// TIA Portal project "Phiva_v4" (V17)

(* hardware
DEVICE "S71500/ET200MP station_1"  S7-1500 station
   slot 0: "Rail_0"  Rack  6ES7 590-1***0-0AA0
   slot 1: "station_1"  CPU 1512C-1 PN  6ES7 512-1CK01-0AB0  V2.5
      slot 3: "CPU display_1"  6ES7591-1AA00-0AA0
      slot 32768: "PROFINET interface_1"  X1
         slot 32769: "Port_1"  X1 P1
         slot 32770: "Port_2"  X1 P2
DEVICE "S71500/ET200MP station_2"  S7-1500 station
   slot 0: "Rail_0"  Rack  6ES7 590-1***0-0AA0
   slot 1: "station_2"  CPU 1512C-1 PN  6ES7 512-1CK01-0AB0  V2.5
      slot 3: "CPU display_1"  6ES7591-1AA00-0AA0
      slot 32768: "PROFINET interface_1"  X1
         slot 32769: "Port_1"  X1 P1
         slot 32770: "Port_2"  X1 P2
DEVICE "HMI_1"  TP700 Comfort
   slot 0: "HMI_1"  TP700 Comfort  6AV2 124-0GC01-0AX0  15.0.0.0
   slot 1: "HMI_RT_1"  TP700 Comfort  6AV2 124-0GC01-0AX0  15.0.0.0
   slot 5: "HMI_1.IE_CP_1"  PROFINET Interface  15.0.0.0
      slot 1: "PROFINET Interface_1"  PROFINET Interface
         slot 1: "Port_1"  Port
         slot 2: "Port_2"  Port
   slot 7: "HMI_1.MPI/DP_CP_1"  MPI/DP Interface  15.0.0.0
*)

// ===== PLC "station_1"  CPU 1512C-1 PN =====

VAR_GLOBAL   // PLC tag table "Default tag table"
   "START" AT %I10.0 : Bool;
   "STOP" AT %I10.1 : Bool;
   "AUTO" AT %I10.2 : Bool;
   "RESET" AT %I10.3 : Bool;
   "START LED" AT %Q4.0 : Bool;
   "RESET LED" AT %Q4.1 : Bool;
   "Q1 LED" AT %Q4.2 : Bool;
   "Q2 LED" AT %Q4.3 : Bool;
   "4 EXTEND PUSH CYLINDER" AT %Q5.4 : Bool;
   "reset_timer_delay_bit" AT %M0.1 : Bool;
   "6 CONVEYOR_1_FORWARD" AT %Q5.0 : Bool;
   "8 INDUCTIVE SENSOR (NO)metal" AT %I11.2 : Bool;
   "7 PART AT DETECTION POSITION(NO)" AT %I11.1 : Bool;
   "5 PUSH CYLINDER EXTENDED" AT %I11.7 : Bool;
   "3 PART IN MAGAZINE (NC)" AT %I11.6 : Bool;
   "power_on_mem" AT %M0.0 : Bool;
   "9 PART AT END CONVEYOR (NO)" AT %I11.0 : Bool;
   "conveyor 2 set active mem" AT %M110.0 : Bool;
   "Tag_1" AT %M200.0 : Bool;
   "System_Byte" AT %MB1 : Byte;
   "FirstScan" AT %M1.0 : Bool;
   "DiagStatusUpdate" AT %M1.1 : Bool;
   "AlwaysTRUE" AT %M1.2 : Bool;
   "AlwaysFALSE" AT %M1.3 : Bool;
   "Clock_Byte" AT %MB500 : Byte;
   "Clock_10Hz" AT %M500.0 : Bool;
   "Clock_5Hz" AT %M500.1 : Bool;
   "Clock_2.5Hz" AT %M500.2 : Bool;
   "Clock_2Hz" AT %M500.3 : Bool;
   "Clock_1.25Hz" AT %M500.4 : Bool;
   "Clock_1Hz" AT %M500.5 : Bool;
   "Clock_0.625Hz" AT %M500.6 : Bool;
   "Clock_0.5Hz" AT %M500.7 : Bool;
   "metal sensor info" AT %M60.0 : Bool;
   "end of conveyor 1" AT %M60.1 : Bool;
   "metal sensor info int" AT %IW60 : Int;
   "any wkpiece info" AT %M80.0 : Bool;
   "station 2 end status" AT %M80.1 : Bool;
   "Tag_2" AT %M70.2 : Bool;
END_VAR

DATA_BLOCK "Data_block_1"   // DB1
{ S7_Optimized_Access := 'FALSE' }
VERSION : 0.1
   VAR
      start_bit : Bool;
      stop_bit : Bool;
      reset_bit : Bool;
      manual_set_bit : Bool;
      power_on_mem : Bool;
      "system_active?" : Bool;
      process_no : Word;
      time_preset : Time := T#2_500MS;
      monitering_time : Time;
      "metal sensor info" : Bool;
      "conveyor 2 status" : Bool;
      "metal sensor info int" : Int;
   END_VAR
BEGIN
END_DATA_BLOCK

DATA_BLOCK "GET"   // DB15
{ S7_Optimized_Access := 'TRUE' }
VERSION : 0.1
   VAR
      GET : Bool;
   END_VAR
BEGIN
END_DATA_BLOCK

// folder: System blocks/Program resources

DATA_BLOCK "reset_button_timer1"   // DB2
{ S7_Optimized_Access := 'TRUE' }
AUTHOR : Simatic
FAMILY : IEC
NAME : IEC_TMR
VERSION : 1.0
// stored: InstanceOfName IEC_TIMER
"IEC_TIMER"
BEGIN
END_DATA_BLOCK

DATA_BLOCK "IEC_Timer_0_DB_2"   // DB3
{ S7_Optimized_Access := 'TRUE' }
AUTHOR : Simatic
FAMILY : IEC
NAME : IEC_TMR
VERSION : 1.0
// stored: InstanceOfName IEC_TIMER
"IEC_TIMER"
BEGIN
END_DATA_BLOCK

DATA_BLOCK "reset_button_timer2"   // DB4
{ S7_Optimized_Access := 'TRUE' }
AUTHOR : Simatic
FAMILY : IEC
NAME : IEC_TMR
VERSION : 1.0
// stored: InstanceOfName IEC_TIMER
"IEC_TIMER"
BEGIN
END_DATA_BLOCK

DATA_BLOCK "IEC_Counter_0_DB"   // DB5
{ S7_Optimized_Access := 'TRUE' }
AUTHOR : Simatic
FAMILY : IEC
NAME : CNTR
VERSION : 1.0
// stored: InstanceOfName IEC_COUNTER
"IEC_COUNTER"
BEGIN
END_DATA_BLOCK

DATA_BLOCK "IEC_Timer_0_DB_3"   // DB6
{ S7_Optimized_Access := 'TRUE' }
AUTHOR : Simatic
FAMILY : IEC
NAME : IEC_TMR
VERSION : 1.0
// stored: InstanceOfName IEC_TIMER
"IEC_TIMER"
BEGIN
END_DATA_BLOCK

DATA_BLOCK "IEC_Counter_0_DB_1"   // DB7
{ S7_Optimized_Access := 'TRUE' }
AUTHOR : Simatic
FAMILY : IEC
NAME : CNTR
VERSION : 1.0
// stored: InstanceOfName IEC_COUNTER
"IEC_COUNTER"
BEGIN
END_DATA_BLOCK

DATA_BLOCK "IEC_Counter_0_DB_2"   // DB8
{ S7_Optimized_Access := 'TRUE' }
AUTHOR : Simatic
FAMILY : IEC
NAME : CNTR
VERSION : 1.0
// stored: InstanceOfName IEC_COUNTER
"IEC_COUNTER"
BEGIN
END_DATA_BLOCK

DATA_BLOCK "reset_time_latch_countdown1"   // DB10
{ S7_Optimized_Access := 'TRUE' }
AUTHOR : Simatic
FAMILY : IEC
NAME : IEC_TMR
VERSION : 1.0
// stored: InstanceOfName IEC_TIMER
"IEC_TIMER"
BEGIN
END_DATA_BLOCK

DATA_BLOCK "IEC_Timer_0_DB"   // DB13
{ S7_Optimized_Access := 'TRUE' }
AUTHOR : Simatic
FAMILY : IEC
NAME : IEC_TMR
VERSION : 1.0
// stored: InstanceOfName IEC_TIMER
"IEC_TIMER"
BEGIN
END_DATA_BLOCK

DATA_BLOCK "IEC_Timer_0_DB_1"   // DB14
{ S7_Optimized_Access := 'TRUE' }
AUTHOR : Simatic
FAMILY : IEC
NAME : IEC_TMR
VERSION : 1.0
// stored: InstanceOfName IEC_TIMER
"IEC_TIMER"
BEGIN
END_DATA_BLOCK

// folder: (top level)

FUNCTION "Auto_Mode" : Void   // FC1, LAD
{ S7_Optimized_Access := 'TRUE' }
VERSION : 0.1
   VAR_TEMP   // added for the SCL form of the ladder/FBD networks
      _w1 : Bool;
      _w2 : Bool;
   END_VAR
BEGIN

REGION Network 1: Detection of material at entry
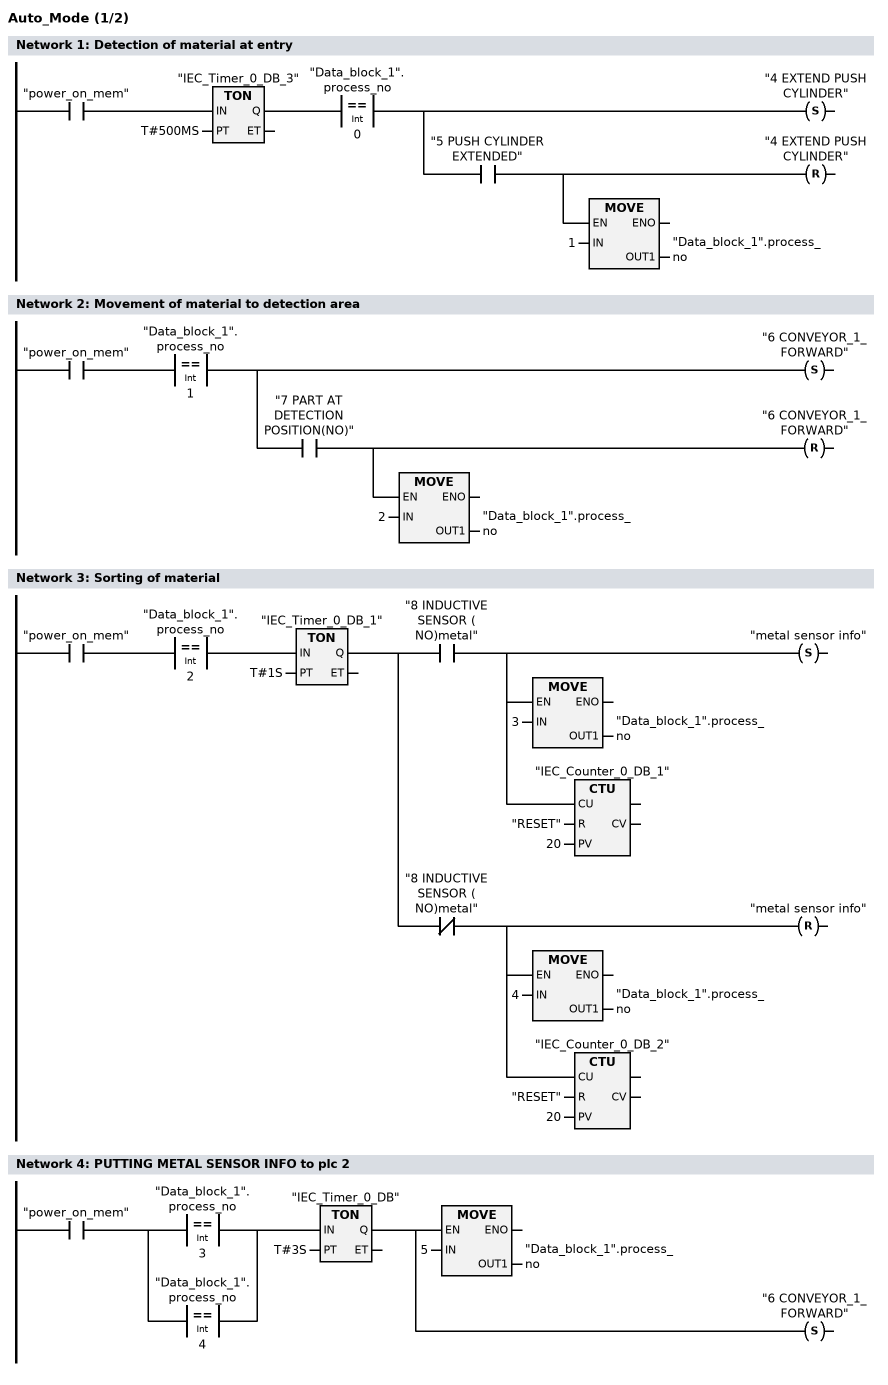
   "IEC_Timer_0_DB_3".TON(IN := "power_on_mem", PT := T#500MS);
   #_w1 := "IEC_Timer_0_DB_3".Q AND ("Data_block_1".process_no = 0);
   IF #_w1 THEN "4 EXTEND PUSH CYLINDER" := TRUE; END_IF;
   IF #_w1 AND "5 PUSH CYLINDER EXTENDED" THEN
       "4 EXTEND PUSH CYLINDER" := FALSE;
       "Data_block_1".process_no := 1;
   END_IF;
END_REGION

REGION Network 2: Movement of material to detection area
   RUNG wire#powerrail
      Contact( "power_on_mem" )
      { S7_Templates := "SrcType := Int" } EQ_Contact(in1 := "Data_block_1".process_no, in2 := 1)
      wire#w1
      S_Coil( "6 CONVEYOR_1_FORWARD" )
   END_RUNG
   RUNG wire#w1
      Contact( "7 PART AT DETECTION POSITION(NO)" )
      wire#w2
      R_Coil( "6 CONVEYOR_1_FORWARD" )
   END_RUNG
   RUNG wire#w2
      Move(in := 2, out1 => "Data_block_1".process_no)
   END_RUNG
   // the same network as SCL:
   #_w1 := "power_on_mem" AND ("Data_block_1".process_no = 1);
   IF #_w1 THEN "6 CONVEYOR_1_FORWARD" := TRUE; END_IF;
   IF #_w1 AND "7 PART AT DETECTION POSITION(NO)" THEN
       "6 CONVEYOR_1_FORWARD" := FALSE;
       "Data_block_1".process_no := 2;
   END_IF;
END_REGION

REGION Network 3: Sorting of material
   "IEC_Timer_0_DB_1".TON(IN := "power_on_mem" AND ("Data_block_1".process_no = 2), PT := T#1S);
   #_w1 := "IEC_Timer_0_DB_1".Q AND "8 INDUCTIVE SENSOR (NO)metal";
   IF #_w1 THEN
       "metal sensor info" := TRUE;
       "Data_block_1".process_no := 3;
   END_IF;
   "IEC_Counter_0_DB_1".CTU(CU := #_w1, R := "RESET", PV := 20);
   #_w2 := "IEC_Timer_0_DB_1".Q AND NOT "8 INDUCTIVE SENSOR (NO)metal";
   IF #_w2 THEN
       "metal sensor info" := FALSE;
       "Data_block_1".process_no := 4;
   END_IF;
   "IEC_Counter_0_DB_2".CTU(CU := #_w2, R := "RESET", PV := 20);
END_REGION

REGION Network 4: PUTTING METAL SENSOR INFO to plc 2
   "IEC_Timer_0_DB".TON(IN := "power_on_mem" AND (("Data_block_1".process_no = 3) OR ("Data_block_1".process_no = 4)),
                        PT := T#3S);
   IF "IEC_Timer_0_DB".Q THEN
       "Data_block_1".process_no := 5;
       "6 CONVEYOR_1_FORWARD" := TRUE;
   END_IF;
END_REGION

REGION Network 5: End of conveyor 1
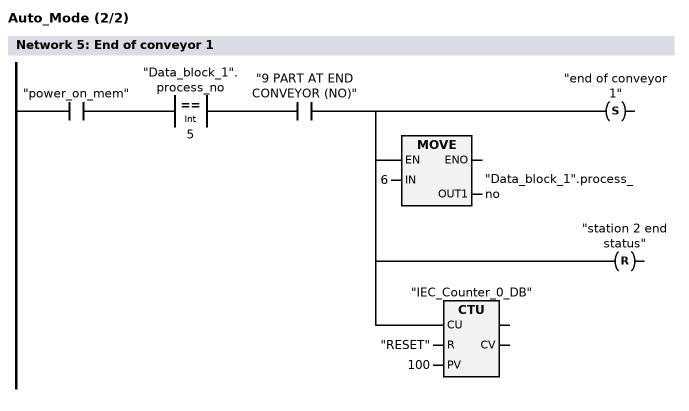
   #_w1 := "power_on_mem" AND ("Data_block_1".process_no = 5) AND "9 PART AT END CONVEYOR (NO)";
   IF #_w1 THEN
       "end of conveyor 1" := TRUE;
       "Data_block_1".process_no := 6;
       "station 2 end status" := FALSE;
   END_IF;
   "IEC_Counter_0_DB".CTU(CU := #_w1, R := "RESET", PV := 100);
END_REGION
END_FUNCTION

FUNCTION "Manual_Mode" : Void   // FC2, LAD
{ S7_Optimized_Access := 'TRUE' }
VERSION : 0.1
BEGIN
END_FUNCTION

ORGANIZATION_BLOCK "Main"   // OB1, LAD, ProgramCycle
TITLE = "Main Program Sweep (Cycle)"
{ S7_Optimized_Access := 'TRUE' }
VERSION : 0.1
   VAR_INPUT
      Initial_Call : Bool;   // Initial call of this OB
      Remanence : Bool;   // =True, if remanent data are available
   END_VAR
   VAR_TEMP   // added for the SCL form of the ladder/FBD networks
      _w1 : Bool;
   END_VAR
BEGIN

REGION Network 1: POWER MEM
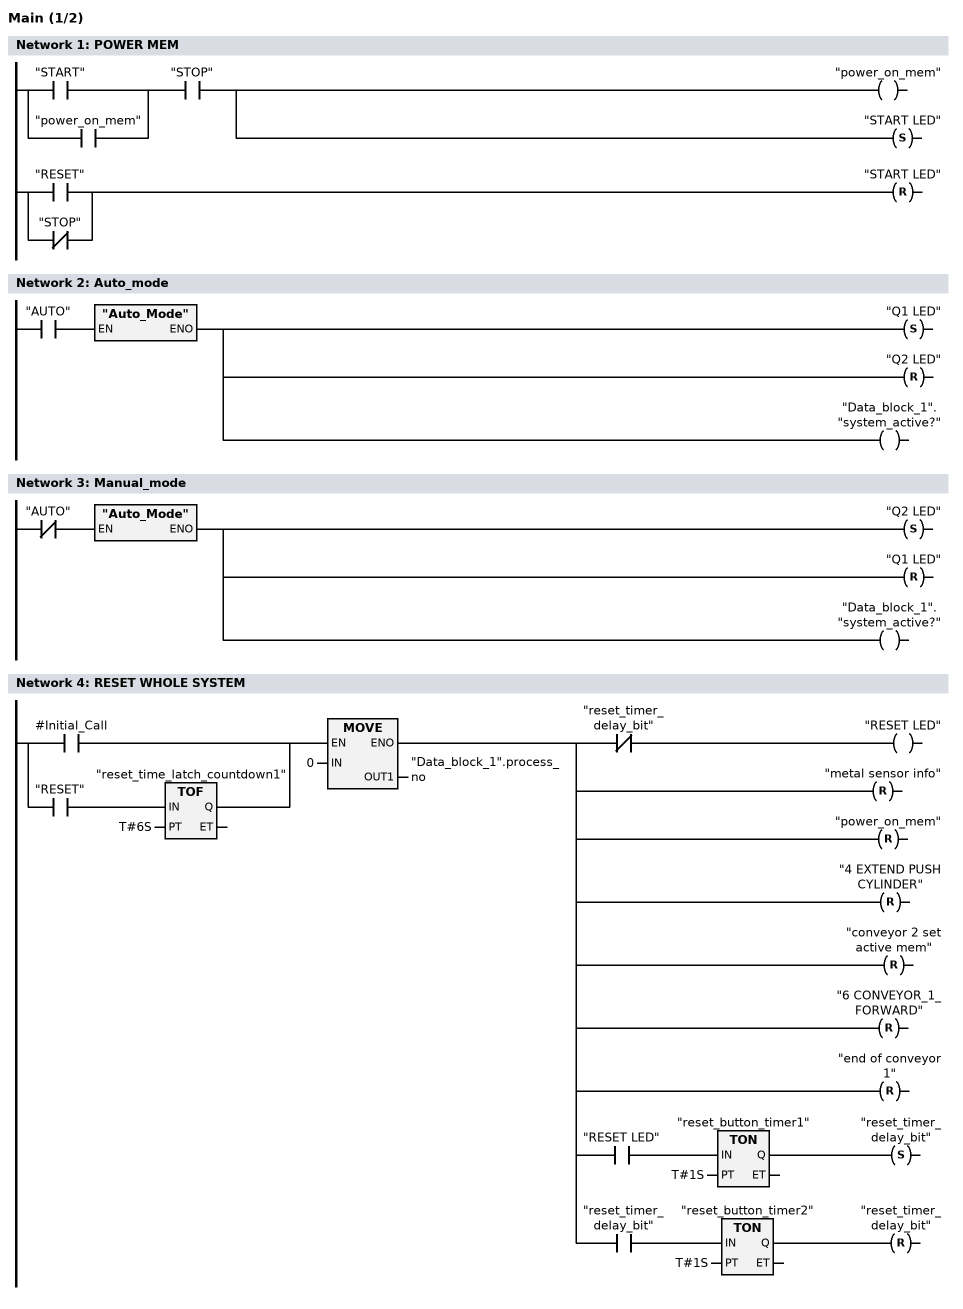
   RUNG wire#powerrail
      Contact( "START" )
      wire#w1
      Contact( "STOP" )
      wire#w2
      Coil( "power_on_mem" )
   END_RUNG
   RUNG wire#powerrail
      Contact( "power_on_mem" )
   END_RUNG wire#w1
   RUNG wire#w2
      S_Coil( "START LED" )
   END_RUNG
   RUNG wire#powerrail
      Contact( "RESET" )
      wire#w3
      R_Coil( "START LED" )
   END_RUNG
   RUNG wire#powerrail
      I_Contact( "STOP" )
   END_RUNG wire#w3
   // the same network as SCL:
   "power_on_mem" := ("START" OR "power_on_mem") AND "STOP";
   IF "power_on_mem" THEN "START LED" := TRUE; END_IF;
   IF "RESET" OR NOT "STOP" THEN "START LED" := FALSE; END_IF;
END_REGION

REGION Network 2: Auto_mode
   RUNG wire#powerrail
      Contact( "AUTO" )
      "Auto_Mode"()
      wire#w1
      S_Coil( "Q1 LED" )
   END_RUNG
   RUNG wire#w1
      R_Coil( "Q2 LED" )
   END_RUNG
   RUNG wire#w1
      Coil( "Data_block_1"."system_active?" )
   END_RUNG
   // the same network as SCL:
   "Auto_Mode"(EN := "AUTO", ENO => #_w1);
   IF #_w1 THEN
       "Q1 LED" := TRUE;
       "Q2 LED" := FALSE;
   END_IF;
   "Data_block_1"."system_active?" := #_w1;
END_REGION

REGION Network 3: Manual_mode
   RUNG wire#powerrail
      I_Contact( "AUTO" )
      "Auto_Mode"()
      wire#w1
      S_Coil( "Q2 LED" )
   END_RUNG
   RUNG wire#w1
      R_Coil( "Q1 LED" )
   END_RUNG
   RUNG wire#w1
      Coil( "Data_block_1"."system_active?" )
   END_RUNG
   // the same network as SCL:
   "Auto_Mode"(EN := NOT "AUTO", ENO => #_w1);
   IF #_w1 THEN
       "Q2 LED" := TRUE;
       "Q1 LED" := FALSE;
   END_IF;
   "Data_block_1"."system_active?" := #_w1;
END_REGION

REGION Network 4: RESET WHOLE SYSTEM
   "reset_time_latch_countdown1".TOF(IN := "RESET", PT := T#6S);
   #_w1 := #Initial_Call OR "reset_time_latch_countdown1".Q;
   IF #_w1 THEN "Data_block_1".process_no := 0; END_IF;
   "RESET LED" := #_w1 AND NOT "reset_timer_delay_bit";
   IF #_w1 THEN
       "metal sensor info" := FALSE;
       "power_on_mem" := FALSE;
       "4 EXTEND PUSH CYLINDER" := FALSE;
       "conveyor 2 set active mem" := FALSE;
       "6 CONVEYOR_1_FORWARD" := FALSE;
       "end of conveyor 1" := FALSE;
   END_IF;
   "reset_button_timer1".TON(IN := #_w1 AND "RESET LED", PT := T#1S);
   IF "reset_button_timer1".Q THEN "reset_timer_delay_bit" := TRUE; END_IF;
   "reset_button_timer2".TON(IN := #_w1 AND "reset_timer_delay_bit", PT := T#1S);
   IF "reset_button_timer2".Q THEN "reset_timer_delay_bit" := FALSE; END_IF;
END_REGION

REGION Network 5: get data from plc 2
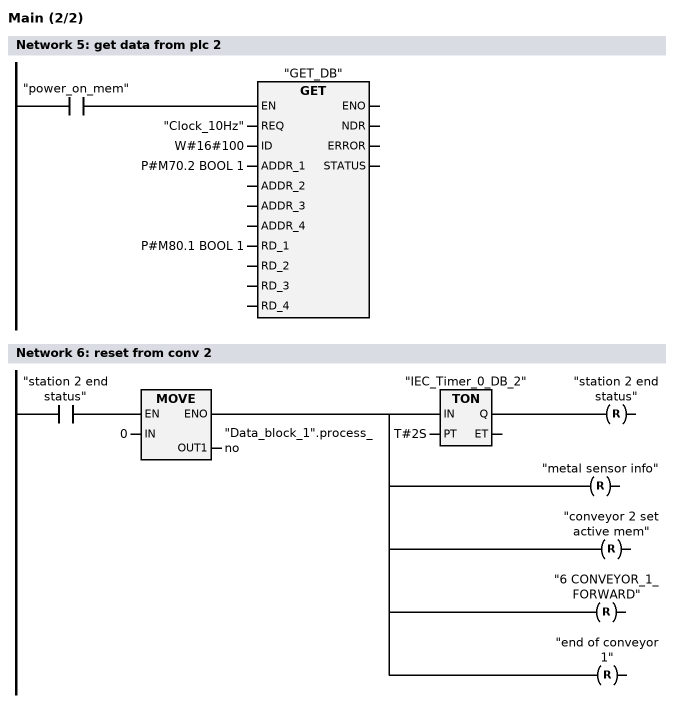
   IF "power_on_mem" THEN
       "GET_DB"(REQ := "Clock_10Hz", ID := W#16#100, ADDR_1 := P#M70.2 BOOL 1, RD_1 := P#M80.1 BOOL 1);   // GET
   END_IF;
END_REGION

REGION Network 6: reset from conv 2
   IF "station 2 end status" THEN "Data_block_1".process_no := 0; END_IF;
   "IEC_Timer_0_DB_2".TON(IN := "station 2 end status", PT := T#2S);
   #_w1 := "station 2 end status";
   IF "IEC_Timer_0_DB_2".Q THEN "station 2 end status" := FALSE; END_IF;
   IF #_w1 THEN
       "metal sensor info" := FALSE;
       "conveyor 2 set active mem" := FALSE;
       "6 CONVEYOR_1_FORWARD" := FALSE;
       "end of conveyor 1" := FALSE;
   END_IF;
END_REGION
END_ORGANIZATION_BLOCK

// ===== PLC "station_2"  CPU 1512C-1 PN =====

VAR_GLOBAL   // PLC tag table "Default tag table"
   "START (NO)" AT %I10.0 : Bool;
   "STOP (NC)" AT %I10.1 : Bool;
   "AUTO" AT %I10.2 : Bool;
   "RESET" AT %I10.3 : Bool;
   "START LED" AT %Q4.0 : Bool;
   "RESET LED" AT %Q4.1 : Bool;
   "Q1 LED" AT %Q4.2 : Bool;
   "Q2 LED" AT %Q4.3 : Bool;
   "8 CONVEYOR 3 FORWARD" AT %Q6.0 : Bool;
   "5 WORKPIECE AT CONVEYOR 2 BARRIER (NC)" AT %I12.0 : Bool;
   "6 CALL ROBOT FOR 2 SEC" AT %Q6.4 : Bool;
   "7 ROBOT DROPPED WORKPIECE AT CONVEYOR 3 (NO)" AT %I12.4 : Bool;
   "9 WORKPIECE EXITING  CONVEYOR 3 (NO)" AT %I12.2 : Bool;
   "3 CONVEYOR 2 FORWARD" AT %Q6.3 : Bool;
   "4 CONVEYOR 2 BARRIER" AT %Q6.2 : Bool;
   "power_on_mem" AT %M0.0 : Bool;
   "6.1 WORKPIECE EXITING STATION 2 (NO)" AT %I12.1 : Bool;
   "non-metal_or_metal_info from plc 1" AT %M70.0 : Bool;
   "Clock_Byte" AT %MB600 : Byte;
   "Clock_10Hz" AT %M600.0 : Bool;
   "Clock_5Hz" AT %M600.1 : Bool;
   "Clock_2.5Hz" AT %M600.2 : Bool;
   "Clock_2Hz" AT %M600.3 : Bool;
   "Clock_1.25Hz" AT %M600.4 : Bool;
   "Clock_1Hz" AT %M600.5 : Bool;
   "Clock_0.625Hz" AT %M600.6 : Bool;
   "Clock_0.5Hz" AT %M600.7 : Bool;
   "reset_timer_delay_bit" AT %M20.0 : Bool;
   "metal sensor info" AT %M20.1 : Bool;
   "conveyor 2 set active mem" AT %M20.2 : Bool;
   "Tag_1" AT %M60.1 : Bool;
   "workpiece ready" AT %M70.1 : Bool;
   "conveyor 2 end process" AT %M70.2 : Bool;
END_VAR

DATA_BLOCK "Receive_data_Block_1"   // DB2
{ S7_Optimized_Access := 'FALSE' }
VERSION : 0.1
   VAR
      "non-metal_or_metal_info" : Bool;
   END_VAR
BEGIN
END_DATA_BLOCK

DATA_BLOCK "Data_block_1"   // DB4
{ S7_Optimized_Access := 'FALSE' }
VERSION : 0.1
   VAR
      process_no : Word;
   END_VAR
BEGIN
END_DATA_BLOCK

// folder: System blocks/Program resources

DATA_BLOCK "IEC_Timer_0_DB"   // DB3
{ S7_Optimized_Access := 'TRUE' }
AUTHOR : Simatic
FAMILY : IEC
NAME : IEC_TMR
VERSION : 1.0
// stored: InstanceOfName IEC_TIMER
"IEC_TIMER"
BEGIN
END_DATA_BLOCK

DATA_BLOCK "IEC_Timer_0_DB_1"   // DB5
{ S7_Optimized_Access := 'TRUE' }
AUTHOR : Simatic
FAMILY : IEC
NAME : IEC_TMR
VERSION : 1.0
// stored: InstanceOfName IEC_TIMER
"IEC_TIMER"
BEGIN
END_DATA_BLOCK

DATA_BLOCK "IEC_Timer_0_DB_2"   // DB6
{ S7_Optimized_Access := 'TRUE' }
AUTHOR : Simatic
FAMILY : IEC
NAME : IEC_TMR
VERSION : 1.0
// stored: InstanceOfName IEC_TIMER
"IEC_TIMER"
BEGIN
END_DATA_BLOCK

DATA_BLOCK "IEC_Counter_0_DB"   // DB7
{ S7_Optimized_Access := 'TRUE' }
AUTHOR : Simatic
FAMILY : IEC
NAME : CNTR
VERSION : 1.0
// stored: InstanceOfName IEC_COUNTER
"IEC_COUNTER"
BEGIN
END_DATA_BLOCK

DATA_BLOCK "IEC_Timer_0_DB_3"   // DB8
{ S7_Optimized_Access := 'TRUE' }
AUTHOR : Simatic
FAMILY : IEC
NAME : IEC_TMR
VERSION : 1.0
// stored: InstanceOfName IEC_TIMER
"IEC_TIMER"
BEGIN
END_DATA_BLOCK

DATA_BLOCK "IEC_Timer_0_DB_4"   // DB9
{ S7_Optimized_Access := 'TRUE' }
AUTHOR : Simatic
FAMILY : IEC
NAME : IEC_TMR
VERSION : 1.0
// stored: InstanceOfName IEC_TIMER
"IEC_TIMER"
BEGIN
END_DATA_BLOCK

DATA_BLOCK "IEC_Counter_0_DB_1"   // DB10
{ S7_Optimized_Access := 'TRUE' }
AUTHOR : Simatic
FAMILY : IEC
NAME : CNTR
VERSION : 1.0
// stored: InstanceOfName IEC_COUNTER
"IEC_COUNTER"
BEGIN
END_DATA_BLOCK

DATA_BLOCK "IEC_Timer_0_DB_5"   // DB11
{ S7_Optimized_Access := 'TRUE' }
AUTHOR : Simatic
FAMILY : IEC
NAME : IEC_TMR
VERSION : 1.0
// stored: InstanceOfName IEC_TIMER
"IEC_TIMER"
BEGIN
END_DATA_BLOCK

DATA_BLOCK "IEC_Timer_0_DB_6"   // DB12
{ S7_Optimized_Access := 'TRUE' }
AUTHOR : Simatic
FAMILY : IEC
NAME : IEC_TMR
VERSION : 1.0
// stored: InstanceOfName IEC_TIMER
"IEC_TIMER"
BEGIN
END_DATA_BLOCK

// folder: (top level)

FUNCTION "Auto_mode_plc_2" : Void   // FC1, LAD
{ S7_Optimized_Access := 'TRUE' }
VERSION : 0.1
   VAR_TEMP   // added for the SCL form of the ladder/FBD networks
      _w1 : Bool;
      _w2 : Bool;
   END_VAR
BEGIN

REGION Network 1: workpiece in conveyor 2
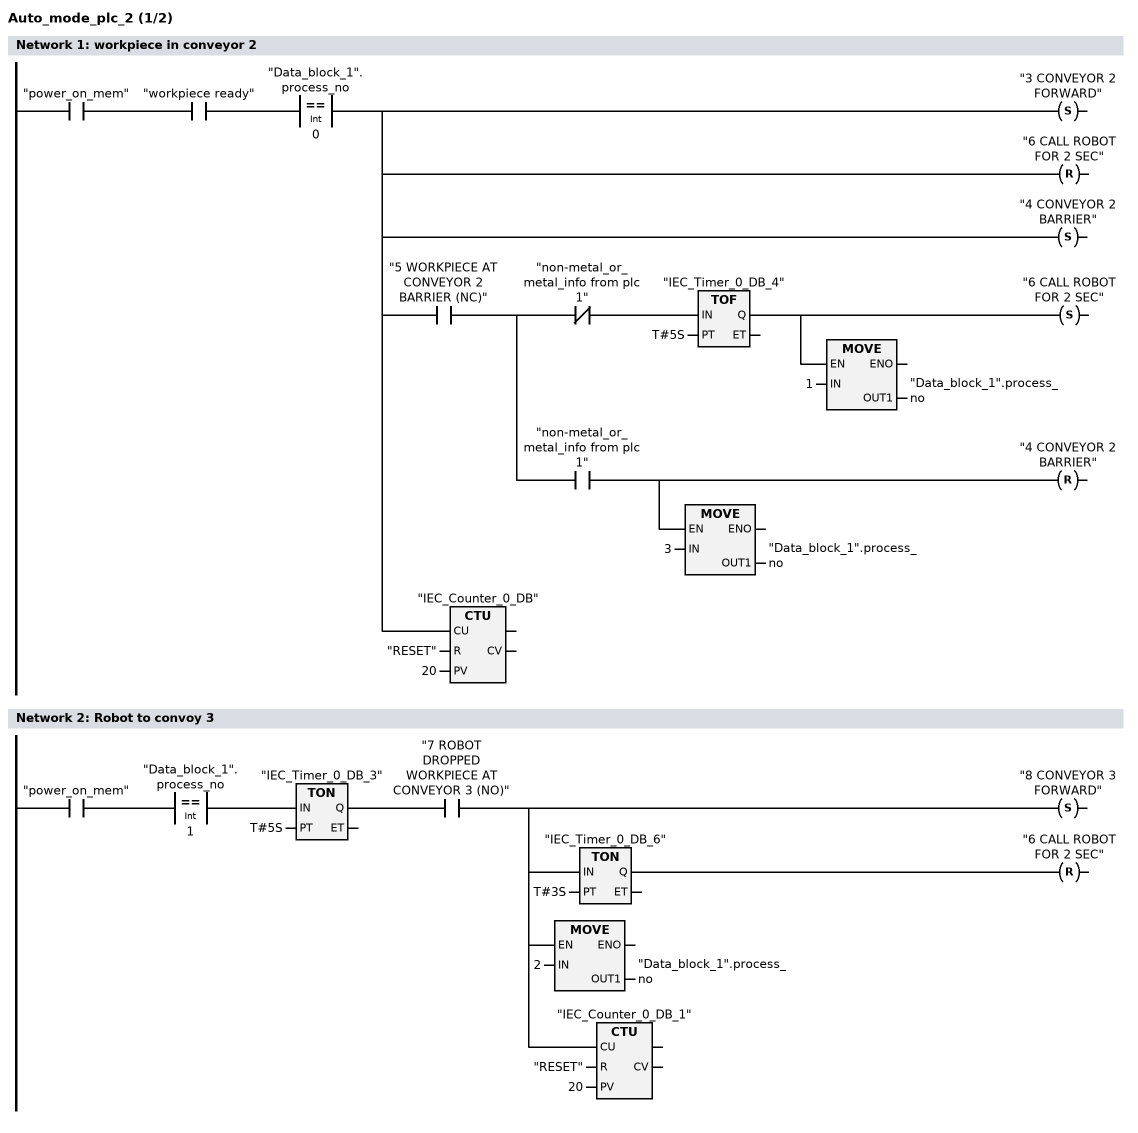
   #_w1 := "power_on_mem" AND "workpiece ready" AND ("Data_block_1".process_no = 0);
   IF #_w1 THEN
       "3 CONVEYOR 2 FORWARD" := TRUE;
       "6 CALL ROBOT FOR 2 SEC" := FALSE;
       "4 CONVEYOR 2 BARRIER" := TRUE;
   END_IF;
   #_w2 := #_w1 AND "5 WORKPIECE AT CONVEYOR 2 BARRIER (NC)";
   "IEC_Timer_0_DB_4".TOF(IN := #_w2 AND NOT "non-metal_or_metal_info from plc 1", PT := T#5S);
   IF "IEC_Timer_0_DB_4".Q THEN
       "6 CALL ROBOT FOR 2 SEC" := TRUE;
       "Data_block_1".process_no := 1;
   END_IF;
   IF #_w2 AND "non-metal_or_metal_info from plc 1" THEN
       "4 CONVEYOR 2 BARRIER" := FALSE;
       "Data_block_1".process_no := 3;
   END_IF;
   "IEC_Counter_0_DB".CTU(CU := #_w1, R := "RESET", PV := 20);
END_REGION

REGION Network 2: Robot to convoy 3
   "IEC_Timer_0_DB_3".TON(IN := "power_on_mem" AND ("Data_block_1".process_no = 1), PT := T#5S);
   #_w1 := "IEC_Timer_0_DB_3".Q AND "7 ROBOT DROPPED WORKPIECE AT CONVEYOR 3 (NO)";
   IF #_w1 THEN "8 CONVEYOR 3 FORWARD" := TRUE; END_IF;
   "IEC_Timer_0_DB_6".TON(IN := #_w1, PT := T#3S);
   IF "IEC_Timer_0_DB_6".Q THEN "6 CALL ROBOT FOR 2 SEC" := FALSE; END_IF;
   IF #_w1 THEN "Data_block_1".process_no := 2; END_IF;
   "IEC_Counter_0_DB_1".CTU(CU := #_w1, R := "RESET", PV := 20);
END_REGION

REGION Network 3: Metal convoyor 3 end + Non-metal exiting station 2
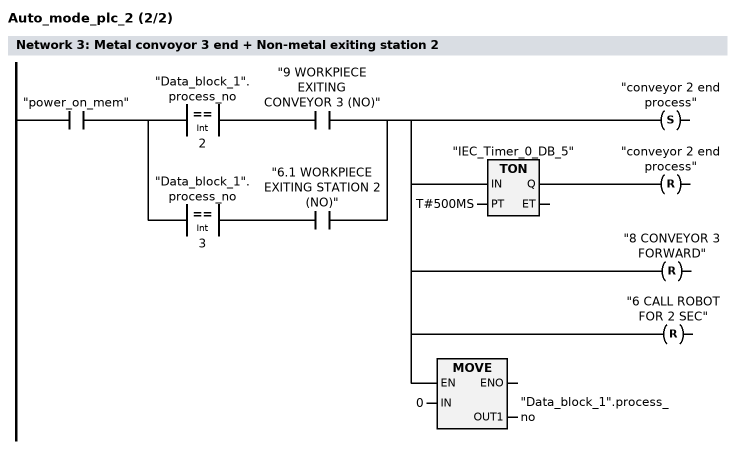
   #_w1 := "power_on_mem" AND ((("Data_block_1".process_no = 2) AND "9 WORKPIECE EXITING  CONVEYOR 3 (NO)") OR (("Data_block_1".process_no = 3) AND "6.1 WORKPIECE EXITING STATION 2 (NO)"));
   IF #_w1 THEN "conveyor 2 end process" := TRUE; END_IF;
   "IEC_Timer_0_DB_5".TON(IN := #_w1, PT := T#500MS);
   IF "IEC_Timer_0_DB_5".Q THEN "conveyor 2 end process" := FALSE; END_IF;
   IF #_w1 THEN
       "8 CONVEYOR 3 FORWARD" := FALSE;
       "6 CALL ROBOT FOR 2 SEC" := FALSE;
       "Data_block_1".process_no := 0;
   END_IF;
END_REGION
END_FUNCTION

FUNCTION "Manual_mode_plc_2" : Void   // FC2, LAD
{ S7_Optimized_Access := 'TRUE' }
VERSION : 0.1
BEGIN
END_FUNCTION

ORGANIZATION_BLOCK "Main"   // OB1, LAD, ProgramCycle
TITLE = "Main Program Sweep (Cycle)"
{ S7_Optimized_Access := 'TRUE' }
VERSION : 0.1
   VAR_INPUT
      Initial_Call : Bool;   // Initial call of this OB
      Remanence : Bool;   // =True, if remanent data are available
   END_VAR
   VAR_TEMP   // added for the SCL form of the ladder/FBD networks
      _w1 : Bool;
   END_VAR
BEGIN

REGION Network 1: POWER MEM
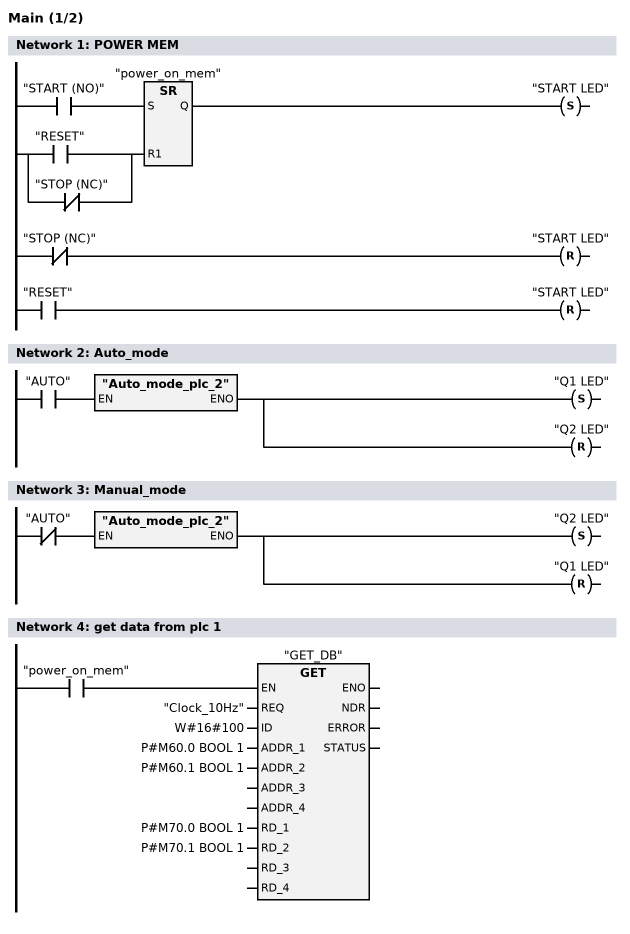
   RUNG wire#powerrail
      Contact( "START (NO)" )
      S_SR(operand := "power_on_mem", r1 := wire#w1)
      S_Coil( "START LED" )
   END_RUNG
   RUNG wire#powerrail
      Contact( "RESET" )
   END_RUNG wire#w1
   RUNG wire#powerrail
      I_Contact( "STOP (NC)" )
   END_RUNG wire#w1
   RUNG wire#powerrail
      I_Contact( "STOP (NC)" )
      R_Coil( "START LED" )
   END_RUNG
   RUNG wire#powerrail
      Contact( "RESET" )
      R_Coil( "START LED" )
   END_RUNG
   // the same network as SCL:
   IF "START (NO)" THEN
       "power_on_mem" := TRUE;   // SR flip-flop
   END_IF;
   IF "RESET" OR NOT "STOP (NC)" THEN "power_on_mem" := FALSE; END_IF;
   IF "power_on_mem" THEN "START LED" := TRUE; END_IF;
   IF NOT "STOP (NC)" THEN "START LED" := FALSE; END_IF;
   IF "RESET" THEN "START LED" := FALSE; END_IF;
END_REGION

REGION Network 2: Auto_mode
   RUNG wire#powerrail
      Contact( "AUTO" )
      "Auto_mode_plc_2"()
      wire#w1
      S_Coil( "Q1 LED" )
   END_RUNG
   RUNG wire#w1
      R_Coil( "Q2 LED" )
   END_RUNG
   // the same network as SCL:
   "Auto_mode_plc_2"(EN := "AUTO", ENO => #_w1);
   IF #_w1 THEN
       "Q1 LED" := TRUE;
       "Q2 LED" := FALSE;
   END_IF;
END_REGION

REGION Network 3: Manual_mode
   RUNG wire#powerrail
      I_Contact( "AUTO" )
      "Auto_mode_plc_2"()
      wire#w1
      S_Coil( "Q2 LED" )
   END_RUNG
   RUNG wire#w1
      R_Coil( "Q1 LED" )
   END_RUNG
   // the same network as SCL:
   "Auto_mode_plc_2"(EN := NOT "AUTO", ENO => #_w1);
   IF #_w1 THEN
       "Q2 LED" := TRUE;
       "Q1 LED" := FALSE;
   END_IF;
END_REGION

REGION Network 4: get data from plc 1
   IF "power_on_mem" THEN
       "GET_DB"(REQ := "Clock_10Hz",   // GET
                ID := W#16#100,
                ADDR_1 := P#M60.0 BOOL 1,
                ADDR_2 := P#M60.1 BOOL 1,
                RD_1 := P#M70.0 BOOL 1,
                RD_2 := P#M70.1 BOOL 1);
   END_IF;
END_REGION

REGION Network 5: RESET WHOLE SYSTEM
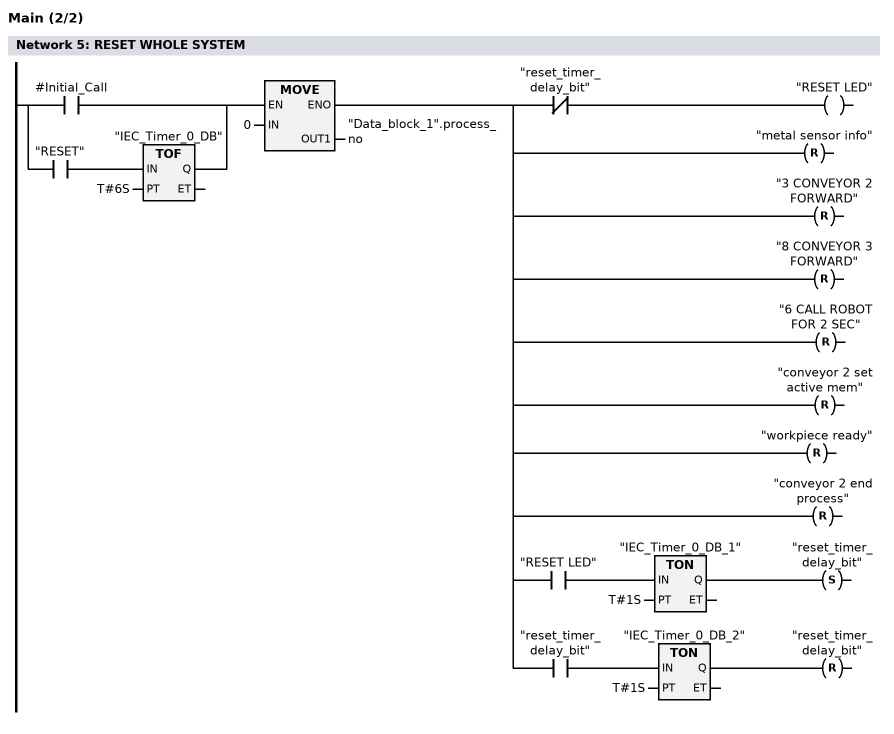
   "IEC_Timer_0_DB".TOF(IN := "RESET", PT := T#6S);
   #_w1 := #Initial_Call OR "IEC_Timer_0_DB".Q;
   IF #_w1 THEN "Data_block_1".process_no := 0; END_IF;
   "RESET LED" := #_w1 AND NOT "reset_timer_delay_bit";
   IF #_w1 THEN
       "metal sensor info" := FALSE;
       "3 CONVEYOR 2 FORWARD" := FALSE;
       "8 CONVEYOR 3 FORWARD" := FALSE;
       "6 CALL ROBOT FOR 2 SEC" := FALSE;
       "conveyor 2 set active mem" := FALSE;
       "workpiece ready" := FALSE;
       "conveyor 2 end process" := FALSE;
   END_IF;
   "IEC_Timer_0_DB_1".TON(IN := #_w1 AND "RESET LED", PT := T#1S);
   IF "IEC_Timer_0_DB_1".Q THEN "reset_timer_delay_bit" := TRUE; END_IF;
   "IEC_Timer_0_DB_2".TON(IN := #_w1 AND "reset_timer_delay_bit", PT := T#1S);
   IF "IEC_Timer_0_DB_2".Q THEN "reset_timer_delay_bit" := FALSE; END_IF;
END_REGION
END_ORGANIZATION_BLOCK

(* ===== HMI "HMI_RT_1" =====
system functions are stored by id; their names below are inferred from use
connection "HMI_Connection_1": ETHERNET, S7_1500_OMS
connection "HMI_Connection_2": ETHERNET, S7_1500_OMS

HMI tags "Default tag table"
   "START" : Bool = PLC START AT %I10.0, 1 s
   "power_on_mem" : Bool = PLC power_on_mem AT %M0.0, 1 s
   "STOP" : Bool = PLC STOP AT %I10.1, 1 s
   "RESET" : Bool = PLC RESET AT %I10.3, 1 s
   "RESET LED" : Bool = PLC "RESET LED" AT %Q4.1, 1 s
   "AUTO" : Bool = PLC AUTO AT %I10.2, 1 s
   "Q1 LED" : Bool = PLC "Q1 LED" AT %Q4.2, 1 s
   "START (NO)" : Bool = PLC "START (NO)" AT %I10.0, 1 s
   "STOP (NC)" : Bool = PLC "STOP (NC)" AT %I10.1, 1 s
   "RESET(1)" : Bool = PLC RESET AT %I10.3, 1 s
   "AUTO(1)" : Bool = PLC AUTO AT %I10.2, 1 s
   "power_on_mem(1)" : Bool = PLC power_on_mem AT %M0.0, 1 s
   "RESET LED(1)" : Bool = PLC "RESET LED" AT %Q4.1, 1 s

screen "Screen_1" 800x480
   Button "Button_1" at 439,20 size 140x43; TextOff 'START BUTTON'
      on Click: SetBit("START (NO)"); ResetBit("STOP (NC)"); ResetBit("RESET(1)")
   Button "Button_2" at 15,20 size 152x37; TextOff 'START BUTTON'
      on Click: SetBit("START"); ResetBit("STOP"); ResetBit("RESET")
   Button "Button_3" at 617,20 size 96x32; TextOff 'STOP'
      on Click: SetBit("STOP (NC)"); ResetBit("START (NO)"); ResetBit("RESET")
   Button "Button_4" at 195,20 size 96x32; TextOff 'STOP'
      on Click: SetBit("STOP"); ResetBit("START")
   Button "Button_5" at 15,173 size 96x62; TextOff 'RESET'
      on Click: SetBit("RESET"); ResetBit("STOP")
   Button "Button_6" at 191,156 size 145x78; TextOff 'MANUAL/AUTO'
      on Click: SetBit("AUTO")
   Button "Button_8" at 617,162 size 159x97; TextOff 'MANUAL/AUTO'
      on Click: SetBit("AUTO(1)")
   Circle "Circle_1" at 15,388 size 91x91
      Appearance <- "Q1 LED"
   TextField "Text field_1" at 15,352 size 63x23; Text 'Q1 LED'
   Circle "Circle_2" at 195,387 size 91x91
      Appearance <- "AUTO"
   Circle "Circle_3" at 617,391 size 83x83
      Appearance <- "AUTO(1)"
   Circle "Circle_4" at 439,395 size 83x83
      Appearance <- "AUTO(1)"
   TextField "Text field_2" at 620,352 size 63x23; Text 'Q2 LED'
   TextField "Text field_3" at 439,360 size 63x23; Text 'Q1 LED'
   TextField "Text field_4" at 204,347 size 63x23; Text 'Q2 LED'
   Circle "Circle_5" at 15,69 size 91x91
      Appearance <- "power_on_mem"
   Circle "Circle_6" at 439,74 size 91x91
      Appearance <- "power_on_mem(1)"
   Circle "Circle_7" at 15,248 size 91x91
      Appearance <- "RESET LED"
   Circle "Circle_8" at 439,265 size 83x83
      Appearance <- "RESET LED(1)"
   Button "Button_7" at 436,190 size 96x32; TextOff 'RESET'
      on Click: SetBit("RESET(1)"); ResetBit("START (NO)"); ResetBit("STOP (NC)")
*)